PROGRAM UN01_StateMachinePallet
VAR
	FB_StateMachineDispenser: FB_StateManager;
	FB_StateMachineShuttle	: FB_StateManager;
	FB_StateMachineOutfeed	: FB_StateManager;
END_VAR

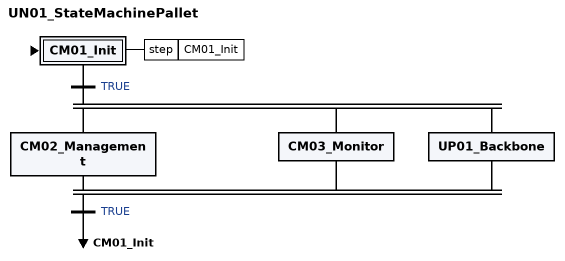
INITIAL_STEP CM01_Init:
    CM01_Init(N);  // step action
END_STEP
TRANSITION FROM CM01_Init TO (CM02_Management, CM03_Monitor, UP01_Backbone)
    := TRUE;
END_TRANSITION
STEP CM02_Management:
END_STEP
STEP CM03_Monitor:
END_STEP
STEP UP01_Backbone:
END_STEP
TRANSITION FROM (CM02_Management, CM03_Monitor, UP01_Backbone) TO CM01_Init
    := TRUE;
END_TRANSITION

ACTION CM01_Init:
//Dispenser
Data_GVL.bFL_StartDispenser 		:= Data_GVL.bStartButton OR HMI_GVL.bStartButtonDispenser;
Data_GVL.bFL_StopDispenser 			:= Data_GVL.bStopButton OR HMI_GVL.bStopButtonDispenser;
Data_GVL.bFL_ResetDispenser 		:= Data_GVL.bResetButton OR HMI_GVL.bResetButtonDispenser;
Data_GVL.bFL_AutoManuaModeDispenser := NOT Data_GVL.StateMachineDispenser.Running AND HMI_GVL.bTestModeEnableDispenser;
//Shuttle
Data_GVL.bFL_StartShuttle 			:= Data_GVL.bStartButton OR HMI_GVL.bStartButtonShuttle;
Data_GVL.bFL_StopShuttle 			:= Data_GVL.bStopButton OR HMI_GVL.bStopButtonShuttle;
Data_GVL.bFL_ResetShuttle 			:= Data_GVL.bResetButton OR HMI_GVL.bResetButtonShuttle;
Data_GVL.bFL_AutoManuaModeShuttle 	:= NOT Data_GVL.StateMachineShuttle.Running AND HMI_GVL.bTestModeEnableShuttle;
//Outfeed
Data_GVL.bFL_StartOutfeed 			:= Data_GVL.bStartButton OR HMI_GVL.bStartButtonOutfeed;
Data_GVL.bFL_StopOutfeed 			:= Data_GVL.bStopButton OR HMI_GVL.bStopButtonOutfeed;
Data_GVL.bFL_ResetOutfeed 			:= Data_GVL.bResetButton OR HMI_GVL.bResetButtonOutfeed;
Data_GVL.bFL_AutoManuaModeOutfeed 	:= NOT Data_GVL.StateMachineOutfeed.Running AND HMI_GVL.bTestModeEnableOutfeed;
END_ACTION

ACTION CM02_Management:
// NETWORK 1
END_ACTION

ACTION CM03_Monitor:
// NETWORK 1
END_ACTION

ACTION UP01_Backbone:
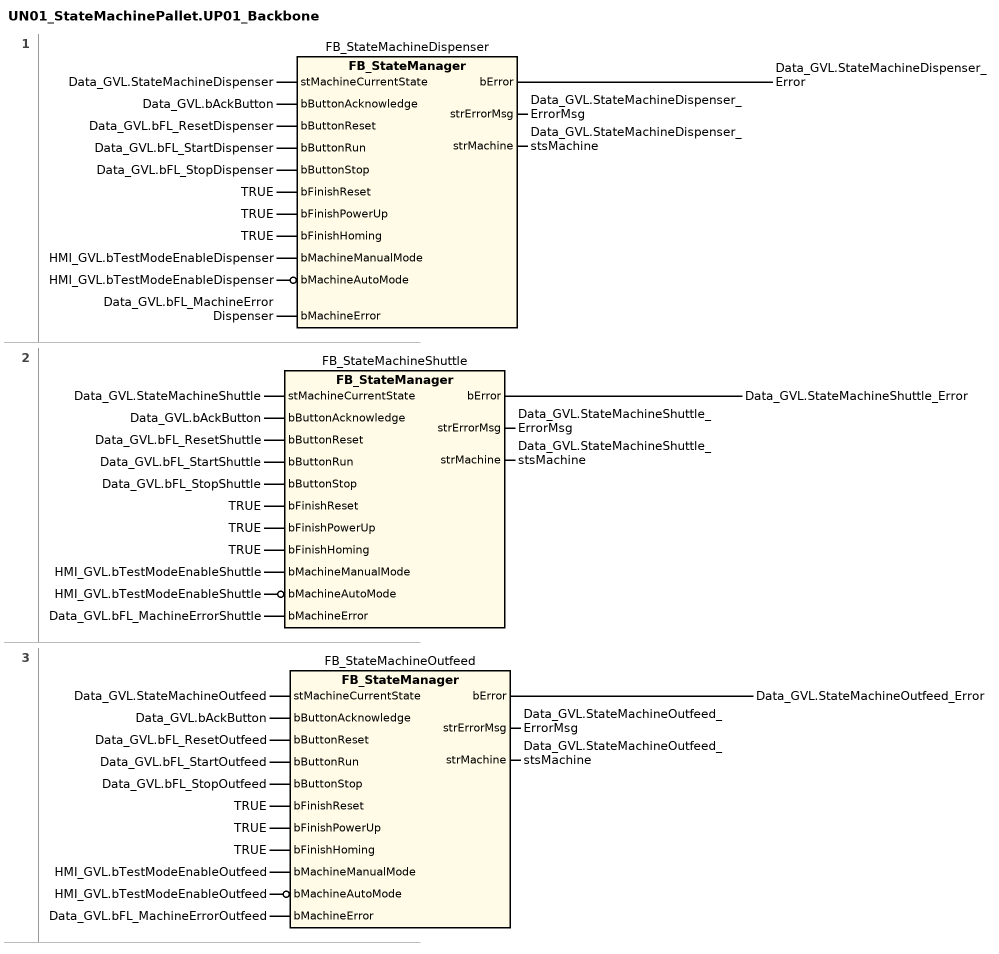
// NETWORK 1
FB_StateMachineDispenser(
    stMachineCurrentState := Data_GVL.StateMachineDispenser,
    bButtonAcknowledge := Data_GVL.bAckButton,
    bButtonReset := Data_GVL.bFL_ResetDispenser,
    bButtonRun := Data_GVL.bFL_StartDispenser,
    bButtonStop := Data_GVL.bFL_StopDispenser,
    bFinishReset := TRUE,
    bFinishPowerUp := TRUE,
    bFinishHoming := TRUE,
    bMachineManualMode := HMI_GVL.bTestModeEnableDispenser,
    bMachineAutoMode := NOT HMI_GVL.bTestModeEnableDispenser,
    bMachineError := Data_GVL.bFL_MachineErrorDispenser,
    strErrorMsg => Data_GVL.StateMachineDispenser_ErrorMsg,
    strMachine => Data_GVL.StateMachineDispenser_stsMachine); // FB_StateManager
Data_GVL.StateMachineDispenser_Error := FB_StateMachineDispenser.bError;

// NETWORK 2
FB_StateMachineShuttle(
    stMachineCurrentState := Data_GVL.StateMachineShuttle,
    bButtonAcknowledge := Data_GVL.bAckButton,
    bButtonReset := Data_GVL.bFL_ResetShuttle,
    bButtonRun := Data_GVL.bFL_StartShuttle,
    bButtonStop := Data_GVL.bFL_StopShuttle,
    bFinishReset := TRUE,
    bFinishPowerUp := TRUE,
    bFinishHoming := TRUE,
    bMachineManualMode := HMI_GVL.bTestModeEnableShuttle,
    bMachineAutoMode := NOT HMI_GVL.bTestModeEnableShuttle,
    bMachineError := Data_GVL.bFL_MachineErrorShuttle,
    strErrorMsg => Data_GVL.StateMachineShuttle_ErrorMsg,
    strMachine => Data_GVL.StateMachineShuttle_stsMachine); // FB_StateManager
Data_GVL.StateMachineShuttle_Error := FB_StateMachineShuttle.bError;

// NETWORK 3
FB_StateMachineOutfeed(
    stMachineCurrentState := Data_GVL.StateMachineOutfeed,
    bButtonAcknowledge := Data_GVL.bAckButton,
    bButtonReset := Data_GVL.bFL_ResetOutfeed,
    bButtonRun := Data_GVL.bFL_StartOutfeed,
    bButtonStop := Data_GVL.bFL_StopOutfeed,
    bFinishReset := TRUE,
    bFinishPowerUp := TRUE,
    bFinishHoming := TRUE,
    bMachineManualMode := HMI_GVL.bTestModeEnableOutfeed,
    bMachineAutoMode := NOT HMI_GVL.bTestModeEnableOutfeed,
    bMachineError := Data_GVL.bFL_MachineErrorOutfeed,
    strErrorMsg => Data_GVL.StateMachineOutfeed_ErrorMsg,
    strMachine => Data_GVL.StateMachineOutfeed_stsMachine); // FB_StateManager
Data_GVL.StateMachineOutfeed_Error := FB_StateMachineOutfeed.bError;
END_ACTION

END_PROGRAM

(* stored: Version 1.1.0.1, ProductVersion 3.1.4024.9
   POU UN01_StateMachinePallet: Id {53203cd3-0102-4694-891f-bfe633260b7c}, SpecialFunc None
   Action CM01_Init: Id {e9626c5e-7689-4ff2-b8e7-e8080edf06fb}
   Action CM02_Management: Id {1d52e868-b823-4e22-90c7-2c9e7fbfcbaa}
   Action CM03_Monitor: Id {b60d57f5-c590-4316-89dd-923699546f35}
   Action UP01_Backbone: Id {55c8013e-88b3-45d8-8d94-c59e6da9d9cf} *)
